// TwinCAT 3 PLC project DAS_A2
// ProgramVersion: 3.1.4020.4
// libraries:
//   Tc2_Standard, * (Beckhoff Automation GmbH)
//   Tc2_System, * (Beckhoff Automation GmbH)
//   Tc3_Module, * (Beckhoff Automation GmbH)
// project tree:
//   DUTs/ ST_PALLET.TcDUT
//   / GlobalTextList.TcGTLO, PlcTask.TcTTO, Visualization Manager.TcVMO (not stored)
//   POUs/ MAIN.TcPOU
//   VISUs/ Visualization.TcVIS
// real-time tasks:
//   TASK PlcTask: cycle T#10ms, priority 20, ADS port 350

CONFIGURATION DAS_A2
    RESOURCE PLC ON TwinCAT3
        TASK PlcTask(INTERVAL := T#10ms, PRIORITY := 20);
        PROGRAM MAIN WITH PlcTask : MAIN;
    END_RESOURCE
END_CONFIGURATION

// ---- DUTs/ST_PALLET.TcDUT
TYPE ST_PALLET :
STRUCT
	WS1: BOOL;
	WS2: BOOL;
	WS3: BOOL;
	FLAG: BOOL:=1;
END_STRUCT
END_TYPE

// ---- POUs/MAIN.TcPOU
PROGRAM MAIN
VAR
	L1: BOOL;
	L2: BOOL;
	L3: BOOL;
	S1: BOOL;
	S2: BOOL;
	S3: BOOL;
	BA1: BOOL;
	BA2: BOOL;
	BA3: BOOL;
	P1: BOOL;
	P2: BOOL;
	P3: BOOL;
	T1: TON;
	T2: TON;
	T3: TON;
	COUNT_IN: INT;
	COUNT_OUT: INT;
	PALLETI: ARRAY [1..50] OF ST_PALLET;
	PALLETV: ARRAY[1..11] OF ST_PALLET;
	I: INT;
	INPUT_PALLET: BOOL;
	INPUT_PALLET_Pressed: BOOL;
	INPUT_PALLET_Released: BOOL;
	INPUT_PALLET_PressedBefore: BOOL;
	StartStop: BOOL;
	MOTOR: BOOL;
	RESET_OUTV1: BOOL;
	RESET_OUTV2: BOOL;
	RESET_OUTV3: BOOL;
	RESET_OUTV4: BOOL;
	RESET_OUTV5: BOOL;
	RESET_OUTV6: BOOL;
	RESET_OUTV7: BOOL;
	RESET_OUTV8: BOOL;
	RESET_OUTV9: BOOL;
	RESET_OUTV10: BOOL;
	RESET_OUTV11: BOOL;
END_VAR

T1(IN:=L1,PT:=T#5S);
T2(IN:=L2,PT:=T#5S);
T3(IN:=L3,PT:=T#5S);

IF INPUT_PALLET_Pressed THEN
	INPUT_PALLET_PressedBefore := TRUE;
ELSIF INPUT_PALLET_Pressed = FALSE AND INPUT_PALLET_PressedBefore THEN
	INPUT_PALLET := TRUE;
	INPUT_PALLET_PressedBefore := FALSE;
END_IF

IF StartStop=FALSE THEN
	MOTOR:=FALSE;
END_IF
//StartStop and input pallet button
IF StartStop THEN
	MOTOR:=TRUE;
	IF INPUT_PALLET AND (COUNT_IN-COUNT_OUT)<11 THEN
	   COUNT_IN:=COUNT_IN +1;
       INPUT_PALLET := FALSE;
    END_IF
//reset memory of output	
	IF RESET_OUTV1 THEN
		PALLETV[1].WS1:=FALSE;
		PALLETV[1].WS2:=FALSE;
		PALLETV[1].WS3:=FALSE;
	END_IF
	IF RESET_OUTV2 THEN
		PALLETV[2].WS1:=FALSE;
		PALLETV[2].WS2:=FALSE;
		PALLETV[2].WS3:=FALSE;
	END_IF
	IF RESET_OUTV3 THEN
		PALLETV[3].WS1:=FALSE;
		PALLETV[3].WS2:=FALSE;
		PALLETV[3].WS3:=FALSE;
	END_IF
	IF RESET_OUTV4 THEN
		PALLETV[4].WS1:=FALSE;
		PALLETV[4].WS2:=FALSE;
		PALLETV[4].WS3:=FALSE;
	END_IF
	IF RESET_OUTV5 THEN
		PALLETV[5].WS1:=FALSE;
		PALLETV[5].WS2:=FALSE;
		PALLETV[5].WS3:=FALSE;
	END_IF
	IF RESET_OUTV6 THEN
		PALLETV[6].WS1:=FALSE;
		PALLETV[6].WS2:=FALSE;
		PALLETV[6].WS3:=FALSE;
	END_IF
	IF RESET_OUTV7 THEN
		PALLETV[7].WS1:=FALSE;
		PALLETV[7].WS2:=FALSE;
		PALLETV[7].WS3:=FALSE;
	END_IF
	IF RESET_OUTV8 THEN
		PALLETV[8].WS1:=FALSE;
		PALLETV[8].WS2:=FALSE;
		PALLETV[8].WS3:=FALSE;
	END_IF
	IF RESET_OUTV9 THEN
		PALLETV[9].WS1:=FALSE;
		PALLETV[9].WS2:=FALSE;
		PALLETV[9].WS3:=FALSE;
	END_IF
	IF RESET_OUTV10 THEN
		PALLETV[10].WS1:=FALSE;
		PALLETV[10].WS2:=FALSE;
		PALLETV[10].WS3:=FALSE;
	END_IF
	IF RESET_OUTV11 THEN
		PALLETV[11].WS1:=FALSE;
		PALLETV[11].WS2:=FALSE;
		PALLETV[11].WS3:=FALSE;
	END_IF
	
	//allocating number to the pallets and reseting finished pallets and also timer reseting
FOR I:=COUNT_IN+1 TO COUNT_IN+1 DO
	IF PALLETI[I].WS1 AND PALLETI[I].WS2 AND PALLETI[I].WS3 THEN
		PALLETV[I]:= PALLETI[I];
		COUNT_OUT:=COUNT_OUT+1;
		PALLETI[I].WS1:=FALSE;
		PALLETI[I].WS2:=FALSE;
		PALLETI[I].WS3:=FALSE;
		PALLETI[I].FLAG:=TRUE;
	END_IF
	IF T1.Q THEN
		L1:=FALSE;
		PALLETI[I].WS1:=TRUE;
		PALLETI[I].FLAG:=TRUE;
	END_IF
	IF T2.Q THEN
		L2:=FALSE;
		PALLETI[I].WS2:=TRUE;
		PALLETI[I].FLAG:=TRUE;
	END_IF	
	IF T3.Q THEN
		L3:=FALSE;
		PALLETI[I].WS3:=TRUE;
		PALLETI[I].FLAG:=TRUE;
	END_IF
	//defining 7*8 different situation that might happen by work stations and tag of the pallets
	IF NOT L1 AND NOT L2 AND NOT L3 THEN
		IF NOT PALLETI[I].WS1 THEN
			IF P1 AND PALLETI[I].FLAG THEN
				S1:=TRUE;
				BA1:=TRUE;
				PALLETI[I].FLAG:=FALSE;
			END_IF
			IF S1 AND BA1 AND L1 THEN
				S1:=FALSE;
				BA1:=FALSE;
			END_IF
		END_IF	
		IF PALLETI[I].WS1 AND NOT PALLETI[I].WS2 AND NOT PALLETI[I].WS3 THEN
			IF P2 AND PALLETI[I].FLAG THEN
				S2:=TRUE;
				BA2:=TRUE;
				P2:=FALSE;
				PALLETI[I].FLAG:=FALSE;
			END_IF
			IF S2 AND BA2 AND L2 THEN
				S2:=FALSE;
				BA2:=FALSE;
			END_IF	
		END_IF
		
		IF PALLETI[I].WS1 AND PALLETI[I].WS2 AND NOT PALLETI[I].WS3 THEN
			IF P3 AND PALLETI[I].FLAG THEN
				S3:=TRUE;
				BA3:=TRUE;
				P3:=FALSE;
				PALLETI[I].FLAG:=FALSE;
			END_IF
			IF S3 AND BA3 AND L3 THEN
				S3:=FALSE;
				BA3:=FALSE;
			END_IF
		END_IF
		IF NOT PALLETI[I].WS1 AND NOT PALLETI[I].WS2 AND PALLETI[I].WS3 THEN
			IF P1 AND PALLETI[I].FLAG THEN
				S1:=TRUE;
				BA1:=TRUE;
				P1:=FALSE;
				PALLETI[I].FLAG:=FALSE;
			END_IF
			IF S1 AND BA1 AND L1 THEN
				S1:=FALSE;
				BA1:=FALSE;
			END_IF
	
			IF P2 AND PALLETI[I].FLAG THEN
				S2:=TRUE;
				BA2:=TRUE;
				P2:=FALSE;
				PALLETI[I].FLAG:=FALSE;
			END_IF
			IF S2 AND BA2 AND L2 THEN
				S2:=FALSE;
				BA2:=FALSE;
			END_IF	
		END_IF	
		IF NOT PALLETI[I].WS1 AND PALLETI[I].WS2 AND PALLETI[I].WS3 THEN
			IF P1 AND PALLETI[I].FLAG THEN
				S1:=TRUE;
				BA1:=TRUE;
				P1:=FALSE;
				PALLETI[I].FLAG:=FALSE;
			END_IF
			IF S1 AND BA1 AND L1 THEN
				S1:=FALSE;
				BA1:=FALSE;
			END_IF
		END_IF	
		IF NOT PALLETI[I].WS1 AND PALLETI[I].WS2 AND NOT PALLETI[I].WS3 THEN
			IF P1 AND PALLETI[I].FLAG THEN
				S1:=TRUE;
				BA1:=TRUE;
				P1:=FALSE;
				PALLETI[I].FLAG:=FALSE;
			END_IF
			IF S1 AND BA1 AND L1 THEN
				S1:=FALSE;
				BA1:=FALSE;
			END_IF
			
			IF P3 AND PALLETI[I].FLAG THEN
				S3:=TRUE;
				BA3:=TRUE;
				P3:=FALSE;
				PALLETI[I].FLAG:=FALSE;
			END_IF
			IF S3 AND BA3 AND L3 THEN
				S3:=FALSE;
				BA3:=FALSE;
			END_IF
		END_IF	
		IF PALLETI[I].WS1 AND NOT PALLETI[I].WS2 AND PALLETI[I].WS3 THEN
			IF P2 AND PALLETI[I].FLAG THEN
				S2:=TRUE;
				BA2:=TRUE;
				P2:=FALSE;
				PALLETI[I].FLAG:=FALSE;
			END_IF
			IF S2 AND BA2 AND L2 THEN
				S2:=FALSE;
				BA2:=FALSE;
			END_IF	
		END_IF	
	END_IF
	IF L1 AND NOT L2 AND NOT L3 THEN
		IF NOT PALLETI[I].WS1 THEN
			IF P1 AND PALLETI[I].FLAG THEN
				S1:=TRUE;
				BA1:=TRUE;
				PALLETI[I].FLAG:=FALSE;
			END_IF
			IF S1 AND BA1 AND L1 THEN
				S1:=FALSE;
				BA1:=FALSE;
			END_IF
		END_IF	
		IF PALLETI[I].WS1 AND NOT PALLETI[I].WS2 AND NOT PALLETI[I].WS3 THEN
			IF P2 AND PALLETI[I].FLAG THEN
				S2:=TRUE;
				BA2:=TRUE;
				P2:=FALSE;
				PALLETI[I].FLAG:=FALSE;
			END_IF
			IF S2 AND BA2 AND L2 THEN
				S2:=FALSE;
				BA2:=FALSE;
			END_IF	
		END_IF	
	
		IF PALLETI[I].WS1 AND PALLETI[I].WS2 AND NOT PALLETI[I].WS3 THEN
			IF P3 AND PALLETI[I].FLAG THEN
				S3:=TRUE;
				BA3:=TRUE;
				P3:=FALSE;
				PALLETI[I].FLAG:=FALSE;
			END_IF
			IF S3 AND BA3 AND L3 THEN
				S3:=FALSE;
				BA3:=FALSE;
			END_IF
		END_IF
		IF NOT PALLETI[I].WS1 AND NOT PALLETI[I].WS2 AND PALLETI[I].WS3 THEN
			IF P1 AND PALLETI[I].FLAG AND NOT L1 THEN
				S1:=TRUE;
				BA1:=TRUE;
				P1:=FALSE;
				PALLETI[I].FLAG:=FALSE;
			END_IF
			IF S1 AND BA1 AND L1 THEN
				S1:=FALSE;
				BA1:=FALSE;
			END_IF
	
			IF P2 AND PALLETI[I].FLAG THEN
				S2:=TRUE;
				BA2:=TRUE;
				P2:=FALSE;
				PALLETI[I].FLAG:=FALSE;
			END_IF
			IF S2 AND BA2 AND L2 THEN
				S2:=FALSE;
				BA2:=FALSE;
			END_IF	
		END_IF	
		IF NOT PALLETI[I].WS1 AND PALLETI[I].WS2 AND PALLETI[I].WS3 THEN
			IF P1 AND PALLETI[I].FLAG AND NOT L1 THEN
				S1:=TRUE;
				BA1:=TRUE;
				P1:=FALSE;
				PALLETI[I].FLAG:=FALSE;
			END_IF
			IF S1 AND BA1 AND L1 THEN
				S1:=FALSE;
				BA1:=FALSE;
			END_IF
		END_IF	
		IF NOT PALLETI[I].WS1 AND PALLETI[I].WS2 AND NOT PALLETI[I].WS3 THEN
			IF P1 AND PALLETI[I].FLAG THEN
				S1:=TRUE;
				BA1:=TRUE;
				P1:=FALSE;
				PALLETI[I].FLAG:=FALSE;
			END_IF
			IF S1 AND BA1 AND L1 THEN
				S1:=FALSE;
				BA1:=FALSE;
			END_IF
			
			IF P3 AND PALLETI[I].FLAG THEN
				S3:=TRUE;
				BA3:=TRUE;
				P3:=FALSE;
				PALLETI[I].FLAG:=FALSE;
			END_IF
			IF S3 AND BA3 AND L3 THEN
				S3:=FALSE;
				BA3:=FALSE;
			END_IF
		END_IF	
		IF PALLETI[I].WS1 AND NOT PALLETI[I].WS2 AND PALLETI[I].WS3 THEN
			IF P2 AND PALLETI[I].FLAG THEN
				S2:=TRUE;
				BA2:=TRUE;
				P2:=FALSE;
				PALLETI[I].FLAG:=FALSE;
			END_IF
			IF S2 AND BA2 AND L2 THEN
				S2:=FALSE;
				BA2:=FALSE;
			END_IF	
		END_IF	
	END_IF
	IF NOT L1 AND L2 AND NOT L3 THEN
		IF NOT PALLETI[I].WS1 THEN
			IF P1 AND PALLETI[I].FLAG THEN
				S1:=TRUE;
				BA1:=TRUE;
				PALLETI[I].FLAG:=FALSE;
			END_IF
			IF S1 AND BA1 AND L1 THEN
				S1:=FALSE;
				BA1:=FALSE;
			END_IF
		END_IF	
		IF PALLETI[I].WS1 AND NOT PALLETI[I].WS2 AND NOT PALLETI[I].WS3 THEN
			IF P2 AND PALLETI[I].FLAG THEN
				S2:=TRUE;
				BA2:=TRUE;
				P2:=FALSE;
				PALLETI[I].FLAG:=FALSE;
			END_IF
			IF S2 AND BA2 AND L2 THEN
				S2:=FALSE;
				BA2:=FALSE;
			END_IF	
		END_IF	
	
		IF PALLETI[I].WS1 AND PALLETI[I].WS2 AND NOT PALLETI[I].WS3 THEN
			IF P3 AND PALLETI[I].FLAG THEN
				S3:=TRUE;
				BA3:=TRUE;
				P3:=FALSE;
				PALLETI[I].FLAG:=FALSE;
			END_IF
			IF S3 AND BA3 AND L3 THEN
				S3:=FALSE;
				BA3:=FALSE;
			END_IF
		END_IF
		IF NOT PALLETI[I].WS1 AND NOT PALLETI[I].WS2 AND PALLETI[I].WS3 THEN
			IF P1 AND PALLETI[I].FLAG AND NOT L1 THEN
				S1:=TRUE;
				BA1:=TRUE;
				P1:=FALSE;
				PALLETI[I].FLAG:=FALSE;
			END_IF
			IF S1 AND BA1 AND L1 THEN
				S1:=FALSE;
				BA1:=FALSE;
			END_IF
	
			IF P2 AND PALLETI[I].FLAG THEN
				S2:=TRUE;
				BA2:=TRUE;
				P2:=FALSE;
				PALLETI[I].FLAG:=FALSE;
			END_IF
			IF S2 AND BA2 AND L2 THEN
				S2:=FALSE;
				BA2:=FALSE;
			END_IF	
		END_IF	
		IF NOT PALLETI[I].WS1 AND PALLETI[I].WS2 AND PALLETI[I].WS3 THEN
			IF P1 AND PALLETI[I].FLAG AND NOT L1 THEN
				S1:=TRUE;
				BA1:=TRUE;
				P1:=FALSE;
				PALLETI[I].FLAG:=FALSE;
			END_IF
			IF S1 AND BA1 AND L1 THEN
				S1:=FALSE;
				BA1:=FALSE;
			END_IF
		END_IF	
		IF NOT PALLETI[I].WS1 AND PALLETI[I].WS2 AND NOT PALLETI[I].WS3 THEN
			IF P1 AND PALLETI[I].FLAG THEN
				S1:=TRUE;
				BA1:=TRUE;
				P1:=FALSE;
				PALLETI[I].FLAG:=FALSE;
			END_IF
			IF S1 AND BA1 AND L1 THEN
				S1:=FALSE;
				BA1:=FALSE;
			END_IF
			
			IF P3 AND PALLETI[I].FLAG THEN
				S3:=TRUE;
				BA3:=TRUE;
				P3:=FALSE;
				PALLETI[I].FLAG:=FALSE;
			END_IF
			IF S3 AND BA3 AND L3 THEN
				S3:=FALSE;
				BA3:=FALSE;
			END_IF
		END_IF	
		IF PALLETI[I].WS1 AND NOT PALLETI[I].WS2 AND PALLETI[I].WS3 THEN
			IF P2 AND PALLETI[I].FLAG THEN
				S2:=TRUE;
				BA2:=TRUE;
				P2:=FALSE;
				PALLETI[I].FLAG:=FALSE;
			END_IF
			IF S2 AND BA2 AND L2 THEN
				S2:=FALSE;
				BA2:=FALSE;
			END_IF	
		END_IF	
	
	END_IF
	IF L1 AND L2 AND NOT L3 THEN
		IF NOT PALLETI[I].WS1 THEN
			IF P1 AND PALLETI[I].FLAG THEN
				S1:=TRUE;
				BA1:=TRUE;
				PALLETI[I].FLAG:=FALSE;
			END_IF
			IF S1 AND BA1 AND L1 THEN
				S1:=FALSE;
				BA1:=FALSE;
			END_IF
		END_IF	
		IF PALLETI[I].WS1 AND NOT PALLETI[I].WS2 AND NOT PALLETI[I].WS3 THEN
			IF P2 AND PALLETI[I].FLAG THEN
				S2:=TRUE;
				BA2:=TRUE;
				P2:=FALSE;
				PALLETI[I].FLAG:=FALSE;
			END_IF
			IF S2 AND BA2 AND L2 THEN
				S2:=FALSE;
				BA2:=FALSE;
			END_IF	
		END_IF	
	
		IF PALLETI[I].WS1 AND PALLETI[I].WS2 AND NOT PALLETI[I].WS3 THEN
			IF P3 AND PALLETI[I].FLAG THEN
				S3:=TRUE;
				BA3:=TRUE;
				P3:=FALSE;
				PALLETI[I].FLAG:=FALSE;
			END_IF
			IF S3 AND BA3 AND L3 THEN
				S3:=FALSE;
				BA3:=FALSE;
			END_IF
		END_IF
		IF NOT PALLETI[I].WS1 AND NOT PALLETI[I].WS2 AND PALLETI[I].WS3 THEN
			IF P1 AND PALLETI[I].FLAG AND NOT L1 THEN
				S1:=TRUE;
				BA1:=TRUE;
				P1:=FALSE;
				PALLETI[I].FLAG:=FALSE;
			END_IF
			IF S1 AND BA1 AND L1 THEN
				S1:=FALSE;
				BA1:=FALSE;
			END_IF
	
			IF P2 AND PALLETI[I].FLAG THEN
				S2:=TRUE;
				BA2:=TRUE;
				P2:=FALSE;
				PALLETI[I].FLAG:=FALSE;
			END_IF
			IF S2 AND BA2 AND L2 THEN
				S2:=FALSE;
				BA2:=FALSE;
			END_IF	
		END_IF	
		IF NOT PALLETI[I].WS1 AND PALLETI[I].WS2 AND PALLETI[I].WS3 THEN
			IF P1 AND PALLETI[I].FLAG AND NOT L1 THEN
				S1:=TRUE;
				BA1:=TRUE;
				P1:=FALSE;
				PALLETI[I].FLAG:=FALSE;
			END_IF
			IF S1 AND BA1 AND L1 THEN
				S1:=FALSE;
				BA1:=FALSE;
			END_IF
		END_IF	
		IF NOT PALLETI[I].WS1 AND PALLETI[I].WS2 AND NOT PALLETI[I].WS3 THEN
			IF P1 AND PALLETI[I].FLAG THEN
				S1:=TRUE;
				BA1:=TRUE;
				P1:=FALSE;
				PALLETI[I].FLAG:=FALSE;
			END_IF
			IF S1 AND BA1 AND L1 THEN
				S1:=FALSE;
				BA1:=FALSE;
			END_IF
			
			IF P3 AND PALLETI[I].FLAG THEN
				S3:=TRUE;
				BA3:=TRUE;
				P3:=FALSE;
				PALLETI[I].FLAG:=FALSE;
			END_IF
			IF S3 AND BA3 AND L3 THEN
				S3:=FALSE;
				BA3:=FALSE;
			END_IF
		END_IF	
		IF PALLETI[I].WS1 AND NOT PALLETI[I].WS2 AND PALLETI[I].WS3 THEN
			IF P2 AND PALLETI[I].FLAG THEN
				S2:=TRUE;
				BA2:=TRUE;
				P2:=FALSE;
				PALLETI[I].FLAG:=FALSE;
			END_IF
			IF S2 AND BA2 AND L2 THEN
				S2:=FALSE;
				BA2:=FALSE;
			END_IF	
		END_IF	
	
	END_IF
	IF NOT L1 AND NOT L2 AND L3 THEN
		IF NOT PALLETI[I].WS1 THEN
			IF P1 AND PALLETI[I].FLAG THEN
				S1:=TRUE;
				BA1:=TRUE;
				PALLETI[I].FLAG:=FALSE;
			END_IF
			IF S1 AND BA1 AND L1 THEN
				S1:=FALSE;
				BA1:=FALSE;
			END_IF
		END_IF	
		IF PALLETI[I].WS1 AND NOT PALLETI[I].WS2 AND NOT PALLETI[I].WS3 THEN
			IF P2 AND PALLETI[I].FLAG THEN
				S2:=TRUE;
				BA2:=TRUE;
				P2:=FALSE;
				PALLETI[I].FLAG:=FALSE;
			END_IF
			IF S2 AND BA2 AND L2 THEN
				S2:=FALSE;
				BA2:=FALSE;
			END_IF	
		END_IF	
	
		IF PALLETI[I].WS1 AND PALLETI[I].WS2 AND NOT PALLETI[I].WS3 THEN
			IF P3 AND PALLETI[I].FLAG THEN
				S3:=TRUE;
				BA3:=TRUE;
				P3:=FALSE;
				PALLETI[I].FLAG:=FALSE;
			END_IF
			IF S3 AND BA3 AND L3 THEN
				S3:=FALSE;
				BA3:=FALSE;
			END_IF
		END_IF
		IF NOT PALLETI[I].WS1 AND NOT PALLETI[I].WS2 AND PALLETI[I].WS3 THEN
			IF P1 AND PALLETI[I].FLAG AND NOT L1 THEN
				S1:=TRUE;
				BA1:=TRUE;
				P1:=FALSE;
				PALLETI[I].FLAG:=FALSE;
			END_IF
			IF S1 AND BA1 AND L1 THEN
				S1:=FALSE;
				BA1:=FALSE;
			END_IF
	
			IF P2 AND PALLETI[I].FLAG THEN
				S2:=TRUE;
				BA2:=TRUE;
				P2:=FALSE;
				PALLETI[I].FLAG:=FALSE;
			END_IF
			IF S2 AND BA2 AND L2 THEN
				S2:=FALSE;
				BA2:=FALSE;
			END_IF	
		END_IF	
		IF NOT PALLETI[I].WS1 AND PALLETI[I].WS2 AND PALLETI[I].WS3 THEN
			IF P1 AND PALLETI[I].FLAG AND NOT L1 THEN
				S1:=TRUE;
				BA1:=TRUE;
				P1:=FALSE;
				PALLETI[I].FLAG:=FALSE;
			END_IF
			IF S1 AND BA1 AND L1 THEN
				S1:=FALSE;
				BA1:=FALSE;
			END_IF
		END_IF	
		IF NOT PALLETI[I].WS1 AND PALLETI[I].WS2 AND NOT PALLETI[I].WS3 THEN
			IF P1 AND PALLETI[I].FLAG THEN
				S1:=TRUE;
				BA1:=TRUE;
				P1:=FALSE;
				PALLETI[I].FLAG:=FALSE;
			END_IF
			IF S1 AND BA1 AND L1 THEN
				S1:=FALSE;
				BA1:=FALSE;
			END_IF
			
			IF P3 AND PALLETI[I].FLAG THEN
				S3:=TRUE;
				BA3:=TRUE;
				P3:=FALSE;
				PALLETI[I].FLAG:=FALSE;
			END_IF
			IF S3 AND BA3 AND L3 THEN
				S3:=FALSE;
				BA3:=FALSE;
			END_IF
		END_IF	
		IF PALLETI[I].WS1 AND NOT PALLETI[I].WS2 AND PALLETI[I].WS3 THEN
			IF P2 AND PALLETI[I].FLAG THEN
				S2:=TRUE;
				BA2:=TRUE;
				P2:=FALSE;
				PALLETI[I].FLAG:=FALSE;
			END_IF
			IF S2 AND BA2 AND L2 THEN
				S2:=FALSE;
				BA2:=FALSE;
			END_IF	
		END_IF	
	
	END_IF	
	IF L1 AND NOT L2 AND L3 THEN
		IF NOT PALLETI[I].WS1 THEN
			IF P1 AND PALLETI[I].FLAG THEN
				S1:=TRUE;
				BA1:=TRUE;
				PALLETI[I].FLAG:=FALSE;
			END_IF
			IF S1 AND BA1 AND L1 THEN
				S1:=FALSE;
				BA1:=FALSE;
			END_IF
		END_IF	
		IF PALLETI[I].WS1 AND NOT PALLETI[I].WS2 AND NOT PALLETI[I].WS3 THEN
			IF P2 AND PALLETI[I].FLAG THEN
				S2:=TRUE;
				BA2:=TRUE;
				P2:=FALSE;
				PALLETI[I].FLAG:=FALSE;
			END_IF
			IF S2 AND BA2 AND L2 THEN
				S2:=FALSE;
				BA2:=FALSE;
			END_IF	
		END_IF	
	
		IF PALLETI[I].WS1 AND PALLETI[I].WS2 AND NOT PALLETI[I].WS3 THEN
			IF P3 AND PALLETI[I].FLAG THEN
				S3:=TRUE;
				BA3:=TRUE;
				P3:=FALSE;
				PALLETI[I].FLAG:=FALSE;
			END_IF
			IF S3 AND BA3 AND L3 THEN
				S3:=FALSE;
				BA3:=FALSE;
			END_IF
		END_IF
		IF NOT PALLETI[I].WS1 AND NOT PALLETI[I].WS2 AND PALLETI[I].WS3 THEN
			IF P1 AND PALLETI[I].FLAG AND NOT L1 THEN
				S1:=TRUE;
				BA1:=TRUE;
				P1:=FALSE;
				PALLETI[I].FLAG:=FALSE;
			END_IF
			IF S1 AND BA1 AND L1 THEN
				S1:=FALSE;
				BA1:=FALSE;
			END_IF
	
			IF P2 AND PALLETI[I].FLAG THEN
				S2:=TRUE;
				BA2:=TRUE;
				P2:=FALSE;
				PALLETI[I].FLAG:=FALSE;
			END_IF
			IF S2 AND BA2 AND L2 THEN
				S2:=FALSE;
				BA2:=FALSE;
			END_IF	
		END_IF	
		IF NOT PALLETI[I].WS1 AND PALLETI[I].WS2 AND PALLETI[I].WS3 THEN
			IF P1 AND PALLETI[I].FLAG AND NOT L1 THEN
				S1:=TRUE;
				BA1:=TRUE;
				P1:=FALSE;
				PALLETI[I].FLAG:=FALSE;
			END_IF
			IF S1 AND BA1 AND L1 THEN
				S1:=FALSE;
				BA1:=FALSE;
			END_IF
		END_IF	
		IF NOT PALLETI[I].WS1 AND PALLETI[I].WS2 AND NOT PALLETI[I].WS3 THEN
			IF P1 AND PALLETI[I].FLAG THEN
				S1:=TRUE;
				BA1:=TRUE;
				P1:=FALSE;
				PALLETI[I].FLAG:=FALSE;
			END_IF
			IF S1 AND BA1 AND L1 THEN
				S1:=FALSE;
				BA1:=FALSE;
			END_IF
			
			IF P3 AND PALLETI[I].FLAG THEN
				S3:=TRUE;
				BA3:=TRUE;
				P3:=FALSE;
				PALLETI[I].FLAG:=FALSE;
			END_IF
			IF S3 AND BA3 AND L3 THEN
				S3:=FALSE;
				BA3:=FALSE;
			END_IF
		END_IF	
		IF PALLETI[I].WS1 AND NOT PALLETI[I].WS2 AND PALLETI[I].WS3 THEN
			IF P2 AND PALLETI[I].FLAG THEN
				S2:=TRUE;
				BA2:=TRUE;
				P2:=FALSE;
				PALLETI[I].FLAG:=FALSE;
			END_IF
			IF S2 AND BA2 AND L2 THEN
				S2:=FALSE;
				BA2:=FALSE;
			END_IF	
		END_IF	
	
	END_IF
	IF NOT L1 AND L2 AND L3 THEN
				IF NOT PALLETI[I].WS1 THEN
			IF P1 AND PALLETI[I].FLAG THEN
				S1:=TRUE;
				BA1:=TRUE;
				PALLETI[I].FLAG:=FALSE;
			END_IF
			IF S1 AND BA1 AND L1 THEN
				S1:=FALSE;
				BA1:=FALSE;
			END_IF
			
		IF PALLETI[I].WS1 AND NOT PALLETI[I].WS2 AND NOT PALLETI[I].WS3 THEN
			IF P2 AND PALLETI[I].FLAG THEN
				S2:=TRUE;
				BA2:=TRUE;
				P2:=FALSE;
				PALLETI[I].FLAG:=FALSE;
			END_IF
			IF S2 AND BA2 AND L2 THEN
				S2:=FALSE;
				BA2:=FALSE;
			END_IF	
		END_IF	
	
		IF PALLETI[I].WS1 AND PALLETI[I].WS2 AND NOT PALLETI[I].WS3 THEN
			IF P3 AND PALLETI[I].FLAG THEN
				S3:=TRUE;
				BA3:=TRUE;
				P3:=FALSE;
				PALLETI[I].FLAG:=FALSE;
			END_IF
			IF S3 AND BA3 AND L3 THEN
				S3:=FALSE;
				BA3:=FALSE;
			END_IF
		END_IF
		IF NOT PALLETI[I].WS1 AND NOT PALLETI[I].WS2 AND PALLETI[I].WS3 THEN
			IF P1 AND PALLETI[I].FLAG AND NOT L1 THEN
				S1:=TRUE;
				BA1:=TRUE;
				P1:=FALSE;
				PALLETI[I].FLAG:=FALSE;
			END_IF
			IF S1 AND BA1 AND L1 THEN
				S1:=FALSE;
				BA1:=FALSE;
			END_IF
	
			IF P2 AND PALLETI[I].FLAG THEN
				S2:=TRUE;
				BA2:=TRUE;
				P2:=FALSE;
				PALLETI[I].FLAG:=FALSE;
			END_IF
			IF S2 AND BA2 AND L2 THEN
				S2:=FALSE;
				BA2:=FALSE;
			END_IF	
		END_IF	
		IF NOT PALLETI[I].WS1 AND PALLETI[I].WS2 AND PALLETI[I].WS3 THEN
			IF P1 AND PALLETI[I].FLAG AND NOT L1 THEN
				S1:=TRUE;
				BA1:=TRUE;
				P1:=FALSE;
				PALLETI[I].FLAG:=FALSE;
			END_IF
			IF S1 AND BA1 AND L1 THEN
				S1:=FALSE;
				BA1:=FALSE;
			END_IF
		END_IF	
		IF NOT PALLETI[I].WS1 AND PALLETI[I].WS2 AND NOT PALLETI[I].WS3 THEN
			IF P1 AND PALLETI[I].FLAG THEN
				S1:=TRUE;
				BA1:=TRUE;
				P1:=FALSE;
				PALLETI[I].FLAG:=FALSE;
			END_IF
			IF S1 AND BA1 AND L1 THEN
				S1:=FALSE;
				BA1:=FALSE;
			END_IF
			
			IF P3 AND PALLETI[I].FLAG THEN
				S3:=TRUE;
				BA3:=TRUE;
				P3:=FALSE;
				PALLETI[I].FLAG:=FALSE;
			END_IF
			IF S3 AND BA3 AND L3 THEN
				S3:=FALSE;
				BA3:=FALSE;
			END_IF
		END_IF	
		IF PALLETI[I].WS1 AND NOT PALLETI[I].WS2 AND PALLETI[I].WS3 THEN
			IF P2 AND PALLETI[I].FLAG THEN
				S2:=TRUE;
				BA2:=TRUE;
				P2:=FALSE;
				PALLETI[I].FLAG:=FALSE;
			END_IF
			IF S2 AND BA2 AND L2 THEN
				S2:=FALSE;
				BA2:=FALSE;
			END_IF	
		END_IF	
	
	END_IF		
	IF PALLETI[I].WS1 AND PALLETI[I].WS2 AND PALLETI[I].WS3 THEN
		PALLETV[I]:= PALLETI[I];
		COUNT_OUT:=COUNT_OUT+1;
		PALLETI[I].WS1:=FALSE;
		PALLETI[I].WS2:=FALSE;
		PALLETI[I].WS3:=FALSE;
		PALLETI[I].FLAG:=TRUE;
	END_IF
		
    END_IF
END_FOR
END_IF

END_PROGRAM

// ---- GlobalTextList.TcGTLO
TEXTLIST GlobalTextList
  10 = 'BA1'
  8 = 'BA2'
  9 = 'BA3'
  38 = 'EXIT PALLET1'
  45 = 'EXIT PALLET10'
  48 = 'EXIT PALLET11'
  47 = 'EXIT PALLET2'
  46 = 'EXIT PALLET3'
  39 = 'EXIT PALLET4'
  40 = 'EXIT PALLET5'
  41 = 'EXIT PALLET6'
  42 = 'EXIT PALLET7'
  43 = 'EXIT PALLET8'
  44 = 'EXIT PALLET9'
  16 = 'Input Pallet'
  3 = 'L1'
  25 = 'L2'
  4 = 'L3'
  14 = 'Motor'
  7 = 'P1'
  6 = 'P2'
  5 = 'P3'
  26 = 'Pallet 1'
  23 = 'Pallet 10'
  27 = 'Pallet 2'
  18 = 'Pallet 3'
  19 = 'Pallet 4'
  20 = 'Pallet 5'
  22 = 'Pallet 6'
  17 = 'Pallet 7'
  24 = 'Pallet 8'
  21 = 'Pallet 9'
  28 = 'RESET PALLET1'
  35 = 'RESET PALLET10'
  37 = 'RESET PALLET2'
  36 = 'RESET PALLET3'
  29 = 'RESET PALLET4'
  30 = 'RESET PALLET5'
  31 = 'RESET PALLET6'
  32 = 'RESET PALLET7'
  33 = 'RESET PALLET8'
  34 = 'RESET PALLET9'
  15 = 'StartStop'
  11 = 'Stopper1'
  13 = 'Stopper2'
  12 = 'Stopper3'
  0 = 'WS1'
  2 = 'WS2'
  1 = 'WS3'
END_TEXTLIST

// ---- VISUs/Visualization.TcVIS
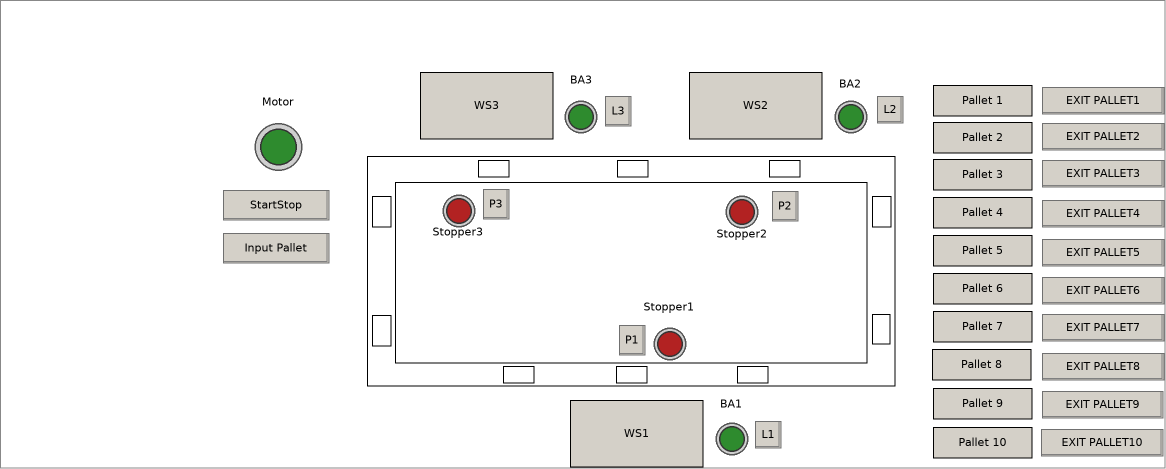
VISUALIZATION Visualization  // 1166x469
    RoundedRectangle (367,156 528x230)
    RoundedRectangle (395,182 472x181)
    Rectangle (570,400 133x67), "WS1", colour toggle: MAIN.T1.Q
    Rectangle (420,72 133x67), "WS3", colour toggle: MAIN.T3.Q
    Rectangle (689,72 133x67), "WS2", colour toggle: MAIN.T2.Q
    Button (755,421 26x27), "L1", text variable: MAIN.L1, colour toggle: MAIN.L1
        toggle MAIN.L1
    Button (605,96 26x30), "L3", text variable: MAIN.L3, colour toggle: MAIN.L3
        toggle MAIN.L3
    Button (483,189 26x30), "P3"
        tap MAIN.P3
    Button (772,191 26x30), "P2"
        tap MAIN.P2
    Button (619,325 26x30), "P1"
        tap MAIN.P1
    Lamp1 (832,94 38x46), tooltip "BA2", variable: MAIN.BA2, style: Lamp-Lamp1-Green
    Label (775,69 150x30), "BA2"
    Lamp1 (562,94 38x46), variable: MAIN.BA3, style: Lamp-Lamp1-Green
    Lamp1 (713,416 38x46), variable: MAIN.BA1, style: Lamp-Lamp1-Green
    Label (506,63 150x34), "BA3"
    Label (656,389 150x30), "BA1"
    Lamp1 (723,189 38x46), variable: MAIN.S2, style: Lamp-Lamp1-Red
    Lamp1 (440,188 38x46), variable: MAIN.S3, style: Lamp-Lamp1-Red
    Lamp1 (651,321 38x46), variable: MAIN.S1, style: Lamp-Lamp1-Red
    Label (594,292 150x30), "Stopper1"
    Label (383,217 150x30), "Stopper3"
    Label (667,219 150x30), "Stopper2"
    Rectangle (503,366 31x17)
    Lamp1 (251,115 55x64), variable: MAIN.MOTOR, style: Lamp-Lamp1-Green
    Label (203,87 150x30), "Motor"
    Button (223,190 106x30), "StartStop"
        toggle MAIN.StartStop
    Button (223,233 106x30), "Input Pallet"
        tap MAIN.INPUT_PALLET_Pressed
    Button (877,96 26x27), "L2", text variable: MAIN.L2, colour toggle: MAIN.L2
        toggle MAIN.L2
    Rectangle (933,85 99x31), "Pallet 1", colour toggle: MAIN.PALLETV[2].WS1
    Rectangle (372,315 19x31)
    Rectangle (617,160 31x17)
    Rectangle (769,160 31x17), invisible if: MAIN.L2
    Rectangle (478,160 31x17), invisible if: MAIN.L3
    Rectangle (737,366 31x17)
    Rectangle (616,366 31x17), invisible if: MAIN.L1
    Rectangle (872,314 18x30)
    Rectangle (872,196 19x31)
    Rectangle (372,196 19x31)
    Rectangle (933,122 99x31), "Pallet 2", colour toggle: MAIN.PALLETV[3].WS1
    Rectangle (933,159 99x31), "Pallet 3", colour toggle: MAIN.PALLETV[4].WS1
    Rectangle (933,197 99x31), "Pallet 4", colour toggle: MAIN.PALLETV[5].WS1
    Rectangle (933,235 99x31), "Pallet 5", colour toggle: MAIN.PALLETV[6].WS1
    Rectangle (933,273 99x31), "Pallet 6", colour toggle: MAIN.PALLETV[7].WS1
    Rectangle (933,311 99x31), "Pallet 7", colour toggle: MAIN.PALLETV[8].WS1
    Rectangle (932,349 99x31), "Pallet 8", colour toggle: MAIN.PALLETV[9].WS1
    Rectangle (933,388 99x31), "Pallet 9", colour toggle: MAIN.PALLETV[10].WS1
    Rectangle (933,427 99x31), "Pallet 10", colour toggle: MAIN.PALLETV[11].WS1
    Button (1041,429 122x27), "EXIT PALLET10"
        tap MAIN.RESET_OUTV11
    Button (1042,160 122x27), "EXIT PALLET3"
        tap MAIN.RESET_OUTV4
    Button (1042,200 122x27), "EXIT PALLET4"
        tap MAIN.RESET_OUTV5
    Button (1042,239 122x27), "EXIT PALLET5"
        tap MAIN.RESET_OUTV6
    Button (1042,277 122x27), "EXIT PALLET6"
        tap MAIN.RESET_OUTV7
    Button (1042,314 122x27), "EXIT PALLET7"
        tap MAIN.RESET_OUTV8
    Button (1042,353 122x27), "EXIT PALLET8"
        tap MAIN.RESET_OUTV9
    Button (1042,391 121x27), "EXIT PALLET9"
        tap MAIN.RESET_OUTV10
    Button (1042,123 122x27), "EXIT PALLET2"
        tap MAIN.RESET_OUTV3
    Button (1042,87 122x27), "EXIT PALLET1"
        tap MAIN.RESET_OUTV2
END_VISUALIZATION
